// TIA Portal V17 export
// export: Created 2024-10-17T14:16:16.8223752Z, ExportSetting WithDefaults, DisplayName Totally Integrated Automation Portal, DisplayVersion V17 Update 4, DisplayName TIA Portal Openness, DisplayVersion V17 Update 4, DisplayName TIA Portal Version Control Interface, DisplayVersion V17, DisplayName SINAMICS Startdrive Advanced, DisplayVersion V17 Update2, DisplayName SINAMICS Startdrive G130, G150, S120, S150, SINAMICS MV, S210, DisplayVersion V17 Update2, DisplayName SINAMICS Startdrive G110M, G120, G120C, G120D, G120P, G115D, DisplayVersion V17 Update2, DisplayName STEP 7 Professional, DisplayVersion V17 Update 4, DisplayName STEP 7 Safety, DisplayVersion V17, DisplayName WinCC Advanced / Unified PC, DisplayVersion V17 Update 4
TYPE "LPMLV2022_typePackTags"
TITLE = LPMLV2022_typePackTags
// Support: tech.team.motioncontrol@siemens.com
// stored: IsFailsafeCompliant false
   STRUCT
      Command : "LPMLV2022_typeCommand";   // Command tags are used to control the operation of the unit/machine. Command tags include unit state commands which control the state transitions in the base state model. The command tags also include parameters and process variables which control how the machine operates
      Status { ExternalWritable := 'False'} : "LPMLV2022_typeStatus";   // Status tags are used to describe the operation of the unit/machine. Status tags include state commands which describe the state transitions in the base state model. The status tags also include parameters and process variables which describe how the machine operates
      Admin { ExternalWritable := 'False'} : "LPMLV2022_typeAdmin";   // Administration tags are used to describe the quality and alarm information of the unit/machine. Administration tags include alarm parameters which describe the conditions within the base state model typically for production data acquisition (PDA) systems. The administration tags also include parameters which can describe how well the machine operates, or specific information on the product quality produced by the machine
   END_STRUCT;
END_TYPE
